TYPE ST_MachineRecipe :
STRUCT
	Station		: ARRAY[0..GVL_StationConfig.nMaxStationCount] OF ST_StationRecipe;
END_STRUCT
END_TYPE

(* stored: Version 1.1.0.1
   DUT ST_MachineRecipe: Id {ecf82cca-35fe-0943-20e4-384f0168efe5} *)
